// Profidrive General State Machine
FUNCTION_BLOCK PUBLIC FB_ProfidriveGSM
VAR_INPUT
	bPowerOn					: BOOL := TRUE;
	bStandstill					: BOOL;
	nControl					: ST_ProfidriveGSM_Control;
END_VAR

VAR_OUTPUT
	nStatus						: ST_ProfidriveGSM_Status;
END_VAR

VAR	
	_eState 					: E_ProfidriveGSM_State := E_ProfidriveGSM_State.S1_SwitchingOnInhibited;
END_VAR

CASE _eState OF 
	E_ProfidriveGSM_State.S0_Disabled : S0_Disabled();
	E_ProfidriveGSM_State.S1_SwitchingOnInhibited : S1_SwitchingOnInhibited();
	E_ProfidriveGSM_State.S2_ReadyForSwitchingOn : S2_ReadyForSwitchingOn();
	E_ProfidriveGSM_State.S3_SwitchedOn : S3_SwitchedOn();
	E_ProfidriveGSM_State.S4_Operation : S4_Operation();
	E_ProfidriveGSM_State.S51_RampStop : S51_RampStop();
	E_ProfidriveGSM_State.S52_QuickStop : S52_QuickStop();
END_CASE

PROPERTY eState : E_ProfidriveGSM_State
GET
eState := _eState;
END_GET
SET
_eState := eState;
END_SET
END_PROPERTY

{ attribute 'hide' }
METHOD PROTECTED S0_Disabled
nStatus.b0_ReadyToSwitchOn 			:= FALSE;				
nStatus.b1_ReadyForOperation 		:= FALSE;				
nStatus.b2_OperationEnabled 		:= FALSE;					
nStatus.b3_FaultPresent 			:= FALSE;						
nStatus.b4_CoastStop 				:= FALSE;	 					
nStatus.b5_QuickStop 				:= FALSE;						
nStatus.b6_SwitchingOnInhibited 	:= FALSE;				
nStatus.b7_WarningPresent			:= FALSE;			
nStatus.b9_ControlRequested 		:= FALSE;	

(*to S1*)	
IF bPowerOn THEN
	_eState := E_ProfidriveGSM_State.S1_SwitchingOnInhibited;
END_IF
END_METHOD

{ attribute 'hide' }
METHOD INTERNAL S1_SwitchingOnInhibited
VAR_INPUT
END_VAR
nStatus.b0_ReadyToSwitchOn 		:= FALSE;				
nStatus.b1_ReadyForOperation 		:= FALSE;				
nStatus.b2_OperationEnabled 		:= FALSE;						
nStatus.b6_SwitchingOnInhibited 	:= TRUE;

(*to S2_ReadyForSwitchingOn*)	
IF NOT nControl.b0_On AND nControl.b1_CoastStop AND nControl.b2_QuickStop THEN
	_eState := E_ProfidriveGSM_State.S2_ReadyForSwitchingOn;
END_IF
END_METHOD

{ attribute 'hide' }
METHOD INTERNAL S2_ReadyForSwitchingOn
VAR_INPUT
END_VAR
nStatus.b0_ReadyToSwitchOn 		:= TRUE;				
nStatus.b1_ReadyForOperation 		:= FALSE;				
nStatus.b2_OperationEnabled 		:= FALSE;						
nStatus.b6_SwitchingOnInhibited 	:= FALSE;

(*to S1_SwitchingOnInhibited*)	
IF NOT nControl.b1_CoastStop OR NOT nControl.b2_QuickStop THEN
	_eState := E_ProfidriveGSM_State.S1_SwitchingOnInhibited;
	RETURN;
END_IF

(*to S3_SwitchedOn*)	
IF nControl.b0_On THEN
	_eState := E_ProfidriveGSM_State.S3_SwitchedOn;
END_IF
END_METHOD

{ attribute 'hide' }
METHOD INTERNAL S3_SwitchedOn
VAR_INPUT
END_VAR
nStatus.b0_ReadyToSwitchOn 		:= TRUE;				
nStatus.b1_ReadyForOperation 		:= TRUE;				
nStatus.b2_OperationEnabled 		:= FALSE;						
nStatus.b6_SwitchingOnInhibited 	:= FALSE;

(*to S1_SwitchingOnInhibited*)	
IF NOT nControl.b1_CoastStop OR NOT nControl.b2_QuickStop THEN
	_eState := E_ProfidriveGSM_State.S1_SwitchingOnInhibited;
	RETURN;
END_IF

(*to S2_ReadyForSwitchingOn*)	
IF NOT nControl.b0_On THEN
	_eState := E_ProfidriveGSM_State.S2_ReadyForSwitchingOn;
	RETURN;
END_IF

(*to S4_Operation*)	
IF nControl.b3_EnableOperation THEN
	_eState := E_ProfidriveGSM_State.S4_Operation;
END_IF
END_METHOD

{ attribute 'hide' }
METHOD INTERNAL S4_Operation
VAR_INPUT
END_VAR
nStatus.b0_ReadyToSwitchOn 		:= TRUE;				
nStatus.b1_ReadyForOperation 		:= TRUE;				
nStatus.b2_OperationEnabled 		:= TRUE;					
nStatus.b6_SwitchingOnInhibited 	:= FALSE;

(*to S1_SwitchingOnInhibited*)	
IF NOT nControl.b1_CoastStop THEN
	_eState := E_ProfidriveGSM_State.S1_SwitchingOnInhibited;
	RETURN;
END_IF

(*to S52_QuickStop*)	
IF NOT nControl.b2_QuickStop THEN
	_eState := E_ProfidriveGSM_State.S52_QuickStop;
	RETURN;
END_IF

(*to S51_RampStop*)	
IF NOT nControl.b0_On THEN
	_eState := E_ProfidriveGSM_State.S51_RampStop;
	RETURN;
END_IF

(*to S3_SwitchedOn*)	
IF NOT nControl.b3_EnableOperation THEN
	_eState := E_ProfidriveGSM_State.S3_SwitchedOn;
END_IF
END_METHOD

{ attribute 'hide' }
METHOD INTERNAL S51_RampStop
VAR_INPUT
END_VAR
nStatus.b0_ReadyToSwitchOn 		:= TRUE;				
nStatus.b1_ReadyForOperation 		:= TRUE;				
nStatus.b2_OperationEnabled 		:= FALSE;					
nStatus.b6_SwitchingOnInhibited 	:= FALSE;

(*to S1_SwitchingOnInhibited*)	
IF NOT nControl.b1_CoastStop THEN
	_eState := E_ProfidriveGSM_State.S1_SwitchingOnInhibited;
	RETURN;
END_IF

(*to S52_QuickStop*)	
IF NOT nControl.b2_QuickStop THEN
	_eState := E_ProfidriveGSM_State.S52_QuickStop;
	RETURN;
END_IF

(*to S2_ReadyForSwitchingOn*)	
IF NOT nControl.b3_EnableOperation OR bStandstill THEN
	_eState := E_ProfidriveGSM_State.S2_ReadyForSwitchingOn;
END_IF

(*to S4_Operation*)	
IF nControl.b0_On THEN
	_eState := E_ProfidriveGSM_State.S4_Operation;
	RETURN;
END_IF
END_METHOD

{ attribute 'hide' }
METHOD INTERNAL S52_QuickStop
VAR_INPUT
END_VAR
nStatus.b0_ReadyToSwitchOn 		:= TRUE;				
nStatus.b1_ReadyForOperation 	:= TRUE;				
nStatus.b2_OperationEnabled 	:= FALSE;					
nStatus.b6_SwitchingOnInhibited := FALSE;

(*to S1_SwitchingOnInhibited*)	
IF NOT nControl.b1_CoastStop THEN
	_eState := E_ProfidriveGSM_State.S1_SwitchingOnInhibited;
	RETURN;
END_IF

(*to S1_SwitchingOnInhibited*)	
IF NOT nControl.b3_EnableOperation OR bStandstill THEN
	_eState := E_ProfidriveGSM_State.S1_SwitchingOnInhibited;
END_IF
END_METHOD

END_FUNCTION_BLOCK

(* stored: Version 1.1.0.1, ProductVersion 3.1.4026.13
   POU FB_ProfidriveGSM: Id {67f99ce3-3e85-0713-170c-0cb2b056b330}, SpecialFunc None
   Property eState: Id {b570af51-38cb-0033-2745-17282cc6abde}
   Get Get: Id {8deb4a10-0007-075c-13d2-4ea7bf51c2c8}
   Set Set: Id {e57f1bbb-544e-0a4e-23ee-f9fbf2a52f32}
   Method S0_Disabled: Id {f7118c5e-d202-0088-1b72-b6ba829282df}
   Method S1_SwitchingOnInhibited: Id {8b1f936f-1181-0c94-2d99-7f7ccdd15167}
   Method S2_ReadyForSwitchingOn: Id {fe11df1e-9b09-052b-2c02-744439a01e9e}
   Method S3_SwitchedOn: Id {440ac6c8-579f-001b-2676-b150543197f5}
   Method S4_Operation: Id {09212b6c-e90e-0497-1e0b-9f10472dcf37}
   Method S51_RampStop: Id {9a23a23b-6923-02b2-3ab0-7ffcb038c1a9}
   Method S52_QuickStop: Id {fe46200a-5223-0841-0e46-ed8ae8fc8e65} *)
